DATA_BLOCK "MotorData"
{ S7_Optimized_Access := 'FALSE' }
VERSION : 0.1
NON_RETAIN
   STRUCT
      Ton {InstructionName := 'TON_TIME'; LibVersion := '1.0'; S7_SetPoint := 'False'} : Array[0..50] of TON_TIME;
      P { S7_SetPoint := 'True'} : Array[0..50] of Bool;
      "Time" : Array[0..50] of Time;
   END_STRUCT;


BEGIN
   "Time"[0] := T#60s;
   "Time"[1] := T#60s;
   "Time"[2] := T#60s;
   "Time"[3] := T#60s;
   "Time"[4] := T#60s;
   "Time"[5] := T#60s;
   "Time"[6] := T#60s;
   "Time"[7] := T#60s;
   "Time"[8] := T#60s;
   "Time"[9] := T#60s;
   "Time"[10] := T#60s;
   "Time"[11] := T#60s;
   "Time"[12] := T#60s;
   "Time"[13] := T#60s;
   "Time"[14] := T#60s;
   "Time"[15] := T#60s;
   "Time"[16] := T#60s;
   "Time"[17] := T#60s;
   "Time"[18] := T#60s;
   "Time"[19] := T#60s;
   "Time"[20] := T#60s;
   "Time"[21] := T#60s;
   "Time"[22] := T#60s;
   "Time"[23] := T#60s;
   "Time"[24] := T#60s;
   "Time"[25] := T#60s;
   "Time"[26] := T#60s;
   "Time"[27] := T#60s;
   "Time"[28] := T#60s;
   "Time"[29] := T#60s;
   "Time"[30] := T#60s;
   "Time"[31] := T#60s;
   "Time"[32] := T#60s;
   "Time"[33] := T#60s;
   "Time"[34] := T#60s;
   "Time"[35] := T#60s;
   "Time"[36] := T#60s;
   "Time"[37] := T#60s;
   "Time"[38] := T#60s;
   "Time"[39] := T#60s;
   "Time"[40] := T#60s;
   "Time"[41] := T#60s;
   "Time"[42] := T#60s;
   "Time"[43] := T#60s;
   "Time"[44] := T#60s;
   "Time"[45] := T#60s;
   "Time"[46] := T#60s;
   "Time"[47] := T#60s;
   "Time"[48] := T#60s;
   "Time"[49] := T#60s;
   "Time"[50] := T#60s;

END_DATA_BLOCK

